TYPE TelemetryDewpointsConfig :
STRUCT
	///Dewpoint of the air at the top of the tube
	topAir: MeasurementConfig;
	///Dewpoint of the air inside the tube
	insideTube: MeasurementConfig;
END_STRUCT
END_TYPE

(* stored: Version 1.1.0.1, ProductVersion 3.1.4019.2
   DUT TelemetryDewpointsConfig: Id {139054e7-df59-4c5a-81bd-7fcc1cec36ca} *)
